# EPICS autosave request: iocBoot/ioc13bma_linux/auto_positions.req
file "Galil_positions.req", P=$(P)
